FUNCTION_BLOCK FB_LamparaTemporizada_IL
VAR_INPUT
    TiempoEncendido: REAL := 2.0;
END_VAR
VAR_OUTPUT
    TiempoPendiente: REAL;
END_VAR
VAR
    Lampara AT %Q*: BOOL;
    Pulsador AT %I*: BOOL;
    
    Temporizador: TON;
    
    Resultado: REAL;
    Tiempo: TIME;
END_VAR

// NETWORK 1
// instruction list
LD      TiempoEncendido
MUL     1000
ST      Resultado

// NETWORK 2
// instruction list
LD      Resultado
REAL_TO_TIME
ST      Tiempo

// NETWORK 3
// instruction list
CAL     Temporizador(
    IN      := Lampara,
    PT      := Tiempo)

// NETWORK 4
// instruction list
LD      Temporizador.ET
TIME_TO_REAL
ST      Resultado

// NETWORK 5
// instruction list
LD      Resultado
DIV     1000
ST      Resultado

// NETWORK 6
// instruction list
LD      TiempoEncendido
SUB     Resultado
ST      TiempoPendiente

// NETWORK 7
// instruction list
LD      Pulsador
S       Lampara

// NETWORK 8
// instruction list
LD      Temporizador.Q
R       Lampara

// NETWORK 9

END_FUNCTION_BLOCK

(* stored: Version 1.1.0.1, ProductVersion 3.1.4024.15
   POU FB_LamparaTemporizada_IL: Id {2efe3ea9-ba30-4661-a60c-8393a923b7df}, SpecialFunc None *)
